TYPE ST_Tension_1 :  //张力FB 接口信号
STRUCT
	fWindDiameter           :REAL;//放卷实时直径
    fDanserDegree           :REAL;//摆杆实时位置
   
   	bTenExecute		        :BOOL;	//张力使能
	bStudyExecute           :BOOL;  //摆杆学习开始     
   	fStudyDiameter          :REAL;  //摆杆学习时放卷直径
	
	bReady                    :BOOL;  //张力功能准备好
	bTensionOK		       :BOOL;	//张力使能OK

	bError			           :BOOL;	//张力出错
                         
END_STRUCT
END_TYPE

(* stored: Version 1.1.0.1, ProductVersion 3.1.4024.12
   DUT ST_Tension_1: Id {6c761de1-8c28-4b7e-9b9f-714e9a3e9ac6} *)
